FUNCTION_BLOCK AxisPowerTestSuite
VAR
	StubAxis : AXIS_REF;
	iStubTask : I_Task;
	TestAxisPower : EnableDisableTask := (AxisRef := StubAxis);
	ObjTestSuite : TestSuite<TestSuiteParameter.MaxTestCount>('C:\ProgramData\Beckhoff\TwinCAT\3.1\Boot\Object_Tests.xml') := (TestSuiteName := 'Object Test Suite');
END_VAR

DoesAxisAcceptEnable_Test();
RejectDisableWhenDisabled_Test();
RejectEnableWhenEnabled_Test();

METHOD DoesAxisAcceptEnable_Test : BOOL
VAR_INST
	Expected : BOOL := TRUE;
	Actual	 : BOOL;
END_VAR
IF ObjTestSuite.Test(__POUNAME()).ExecuteTest() THEN
	Actual := SUCCEEDED(TestAxisPower.Enable());
	TestAxisPower.Disable();
	ObjTestSuite.Test(__POUNAME()).AssertEqual(Expected, Actual);
END_IF
END_METHOD

METHOD RejectDisableWhenDisabled_Test : BOOL
VAR_INST
	Expected : BOOL := TRUE;
	Actual	 : BOOL;
END_VAR
IF ObjTestSuite.Test(__POUNAME()).ExecuteTest() THEN
	Actual := FAILED(TestAxisPower.Disable());
	ObjTestSuite.Test(__POUNAME()).AssertEqual(Expected, Actual);
END_IF
END_METHOD

METHOD RejectEnableWhenEnabled_Test : BOOL
VAR_INST
	Expected : BOOL := TRUE;
	Actual	 : BOOL;
END_VAR
IF ObjTestSuite.Test(__POUNAME()).ExecuteTest() THEN
	TestAxisPower.Enable();
	Actual := FAILED(TestAxisPower.Enable());
	TestAxisPower.Abort();
	ObjTestSuite.Test(__POUNAME()).AssertEqual(Expected, Actual);
END_IF
END_METHOD

END_FUNCTION_BLOCK

(* stored: Version 1.1.0.1
   POU AxisPowerTestSuite: Id {ac2625ce-9cae-4674-bbac-7fb3863ceb8a}, SpecialFunc None
   Method DoesAxisAcceptEnable_Test: Id {fe79904b-ba9b-4299-9251-955ef4cd651f}
   Method RejectDisableWhenDisabled_Test: Id {2c27dff1-a943-4ffc-b0d9-e00a76c5c4af}
   Method RejectEnableWhenEnabled_Test: Id {3a8db93e-7de7-40e7-bc08-d2e3cb8c9735} *)
